SUBAPPLICATION Uebung_111 (* Übung zum Integer Überlauf *)
  (* Standard: 61499-2; Description: Copyright (c) 2023 Meisterschulen am Ostbahnhof This program and the accompanying materials are made available under the terms of the Eclipse Public License 2.0 which is available at https://www.eclipse.org/legal/epl-2.0/ SPDX-License-Identifier: EPL-2.0 *)
  (* Version 1.0, 2023-10-23, Franz Höpfinger, Meisterschulen am Ostbahnhof *)
  PACKAGE Uebungen;
  IMPORT logiBUS::io::DI::logiBUS_DI::Input_I1;
  IMPORT logiBUS::io::DI::logiBUS_DI_Events::BUTTON_SINGLE_CLICK;
  IMPORT logiBUS::io::DQ::logiBUS_DO::Output_Q1;
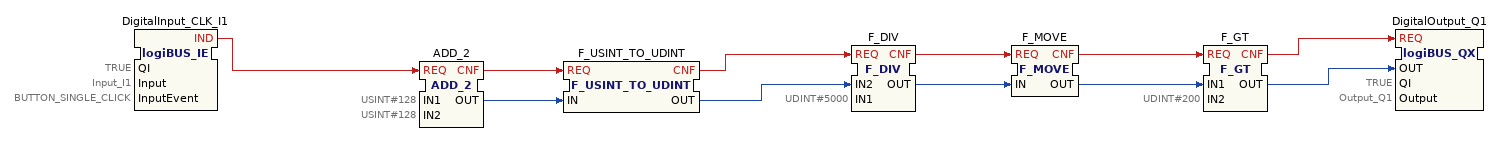
  FBS
    DigitalOutput_Q1 : logiBUS::io::DQ::logiBUS_QX(QI := TRUE, Output := Output_Q1);
    ADD_2 : iec61131::arithmetic::ADD_2(IN1 := USINT#128, IN2 := USINT#128);
    DigitalInput_CLK_I1 : logiBUS::io::DI::logiBUS_IE(QI := TRUE, Input := Input_I1, InputEvent := BUTTON_SINGLE_CLICK);
    F_GT : iec61131::comparison::F_GT(IN2 := UDINT#200);
    F_DIV : iec61131::arithmetic::F_DIV(IN1 := UDINT#5000);
    F_USINT_TO_UDINT : iec61131::conversion::F_USINT_TO_UDINT;
    F_MOVE : iec61131::selection::F_MOVE; {SET_ATTRIBUTE(DataType, UDINT)}
  END_FBS
  EVENT_CONNECTIONS
    DigitalInput_CLK_I1.IND TO ADD_2.REQ;
    F_GT.CNF TO DigitalOutput_Q1.REQ;
    ADD_2.CNF TO F_USINT_TO_UDINT.REQ;
    F_USINT_TO_UDINT.CNF TO F_DIV.REQ;
    F_DIV.CNF TO F_MOVE.REQ;
    F_MOVE.CNF TO F_GT.REQ;
  END_CONNECTIONS
  DATA_CONNECTIONS
    F_GT.OUT TO DigitalOutput_Q1.OUT;
    ADD_2.OUT TO F_USINT_TO_UDINT.IN;
    F_USINT_TO_UDINT.OUT TO F_DIV.IN2;
    F_MOVE.OUT TO F_GT.IN1;
    F_DIV.OUT TO F_MOVE.IN;
  END_CONNECTIONS
END_SUBAPPLICATION
